Staubli VAL3: SETBIT.pgx

public program setBit(num x_bit, num& x_return[])
// set a bit in a num variable
  local num l_mask
begin
  call bmask(x_bit,l_mask)
  x_return=x_return+l_mask
  if bDebug
    putln("setBit(): "+toString("0.0",x_return))
  endIf
end
